# EPICS autosave request: iocBoot/iocDante/auto_settings.req
file "dante_settings.req",        P=$(P), R=$(R)
file "danteN_settings.req",        P=$(P), R=$(R)
file "mca_settings.req",          P=$(P), M=$(M)
file "commonPlugin_settings.req", P=$(P)
